// Mitsubishi GX Works2 project: Pneumalek2   PLC: Q03UDE

// global labels: Global1
VAR_GLOBAL
  Läge_0 AT M0 : BOOL;  (* Sensor *)
  Läge_1 AT M1 : BOOL;  (* Sensor *)
  Mag_sens AT M6 : BOOL;  (* Sensor *)
  Hämta_Mag : BOOL;
  Läge_2 AT M2 : BOOL;  (* Sensor *)
  Vrid_0 AT M3 : BOOL;  (* Sensor *)
  Vrid_1 AT M4 : BOOL;  (* Sensor *)
  Vrid_2 AT M5 : BOOL;  (* Sensor *)
  Kapacitiv AT M7 : BOOL;  (* Sensor *)
  Foto AT M8 : BOOL;  (* Sensor *)
  Induktiv AT M9 : BOOL;  (* Sensor *)
  Vakuum AT M10 : BOOL;  (* Sensor *)
  CylUppe AT M11 : BOOL;  (* Sensor *)
  CylNere AT M12 : BOOL;  (* Sensor *)
  Start AT M14 : BOOL;  (* Sensor *)
  Stopp AT M15 : BOOL;  (* Sensor *)
  PortalUt AT M17 : BOOL;  (* Actuator *)
  PortalIn AT M18 : BOOL;  (* Actuator *)
  VridHöger AT M19 : BOOL;  (* Actuator *)
  VridVänster AT M20 : BOOL;  (* Actuator *)
  CylNer AT M21 : BOOL;  (* Actuator *)
  CylUpp AT M22 : BOOL;  (* Actuator *)
  Sug : BOOL;
  Lämna_Sens : BOOL;
  Metall : BOOL;
  Vit : BOOL;
  Svart : BOOL;
  Sensor_Kopp : BOOL;
  Hämta_Sens : BOOL;
  LämnaMetall : BOOL;
  LämnaSvart : BOOL;
  LämnaVit : BOOL;
  Ejektor AT M23 : BOOL;  (* Actuator *)
  RESET : BOOL;
  ResetLägeP AT M16 : BOOL;  (* Sensor *)
  Portal : INT;
  Vrid : INT;
  PortalPos : INT;
  VridPos : INT;
  Hämta : BOOL;  (* Utan Last *)
  Lämna : BOOL;  (* Med Last *)
  Test_1 : BOOL;
  TestTimer1 : TON;
  TestTimer2 : TON;
  TestTimer3 : TON;
  TestTimer4 : TON;
  TestCount_1 : CTU;
  Testfunk1 : BOOL;
  TestTimer5 : TON;
  TestTimer6 : TON;
  TestTimer7 : TON;
  VridEQ : BOOL;
  PortalEQ : BOOL;
  Vänta_Sens : BOOL;
  TestM : BOOL;
  TestV : BOOL;
  TestS : BOOL;
  TestTimer8 : TON;
  TestTimer9 : TON;
  Timer7 : TON;
END_VAR

// task Task_01 (event TRUE, interval 0, priority 31): Sekvens, Applikation, testa

PROGRAM Sekvens
VAR
  Kör : BOOL;
END_VAR
(* structured ladder/FBD written out as ST: instructions are called as NAME(EN, inputs, outputs); _pN, _eN, _tN stand for wires *)
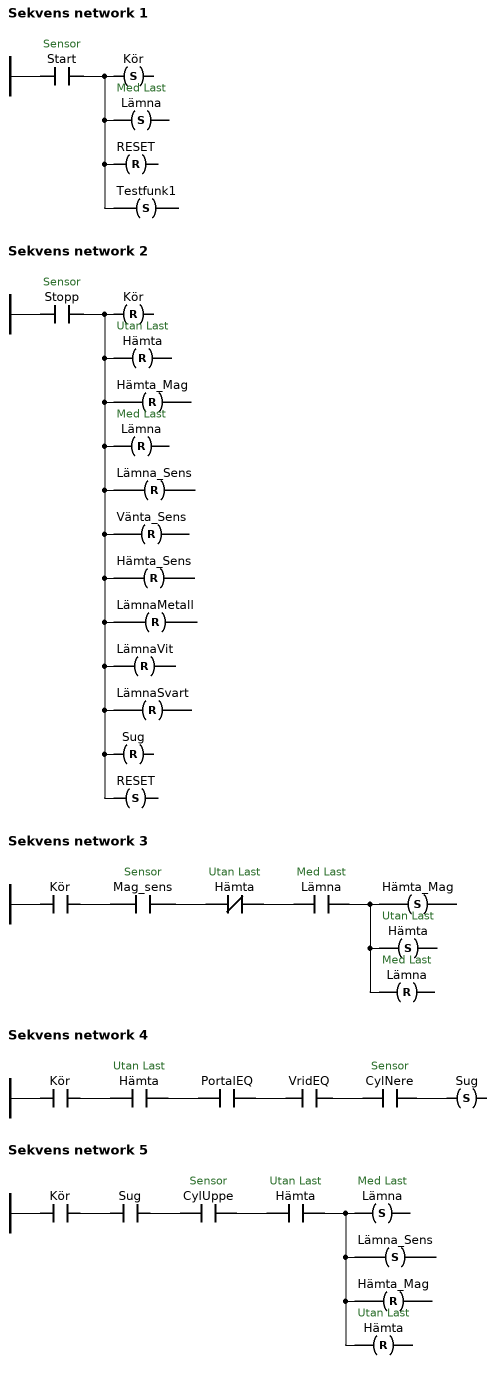
(* network 1 *)
SET(Start, Kör);
SET(Start, Lämna);
RST(Start, RESET);
SET(Start, Testfunk1);
(* network 2 *)
RST(Stopp, Kör);
RST(Stopp, Hämta);
RST(Stopp, Hämta_Mag);
RST(Stopp, Lämna);
RST(Stopp, Lämna_Sens);
RST(Stopp, Vänta_Sens);
RST(Stopp, Hämta_Sens);
RST(Stopp, LämnaMetall);
RST(Stopp, LämnaVit);
RST(Stopp, LämnaSvart);
RST(Stopp, Sug);
SET(Stopp, RESET);
(* network 3 *)
_p1 := Kör AND Mag_sens AND NOT Hämta AND Lämna;
SET(_p1, Hämta_Mag);
SET(_p1, Hämta);
RST(_p1, Lämna);
(* network 4 *)
SET(Kör AND Hämta AND PortalEQ AND VridEQ AND CylNere, Sug);
(* network 5 *)
_p1 := Kör AND Sug AND CylUppe AND Hämta;
SET(_p1, Lämna);
SET(_p1, Lämna_Sens);
RST(_p1, Hämta_Mag);
RST(_p1, Hämta);
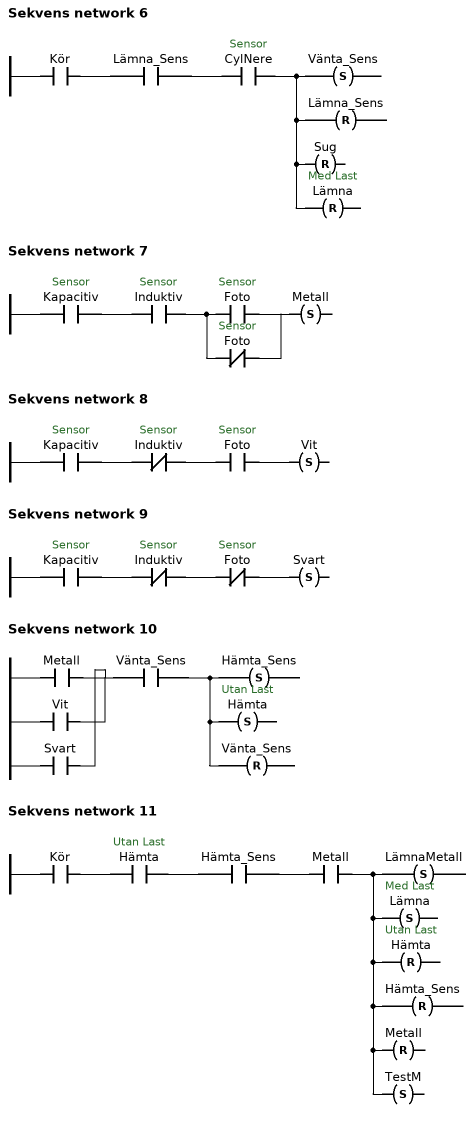
(* network 6 *)
_p1 := Kör AND Lämna_Sens AND CylNere;
SET(_p1, Vänta_Sens);
RST(_p1, Lämna_Sens);
RST(_p1, Sug);
RST(_p1, Lämna);
(* network 7 *)
_p1 := Kapacitiv AND Induktiv;
SET((_p1 AND Foto) OR (_p1 AND NOT Foto), Metall);
(* network 8 *)
SET(Kapacitiv AND NOT Induktiv AND Foto, Vit);
(* network 9 *)
SET(Kapacitiv AND NOT Induktiv AND NOT Foto, Svart);
(* network 10 *)
_p1 := (Metall OR Vit OR Svart) AND Vänta_Sens;
SET(_p1, Hämta_Sens);
SET(_p1, Hämta);
RST(_p1, Vänta_Sens);
(* network 11 *)
_p1 := Kör AND Hämta AND Hämta_Sens AND Metall;
SET(_p1, LämnaMetall);
SET(_p1, Lämna);
RST(_p1, Hämta);
RST(_p1, Hämta_Sens);
RST(_p1, Metall);
SET(_p1, TestM);
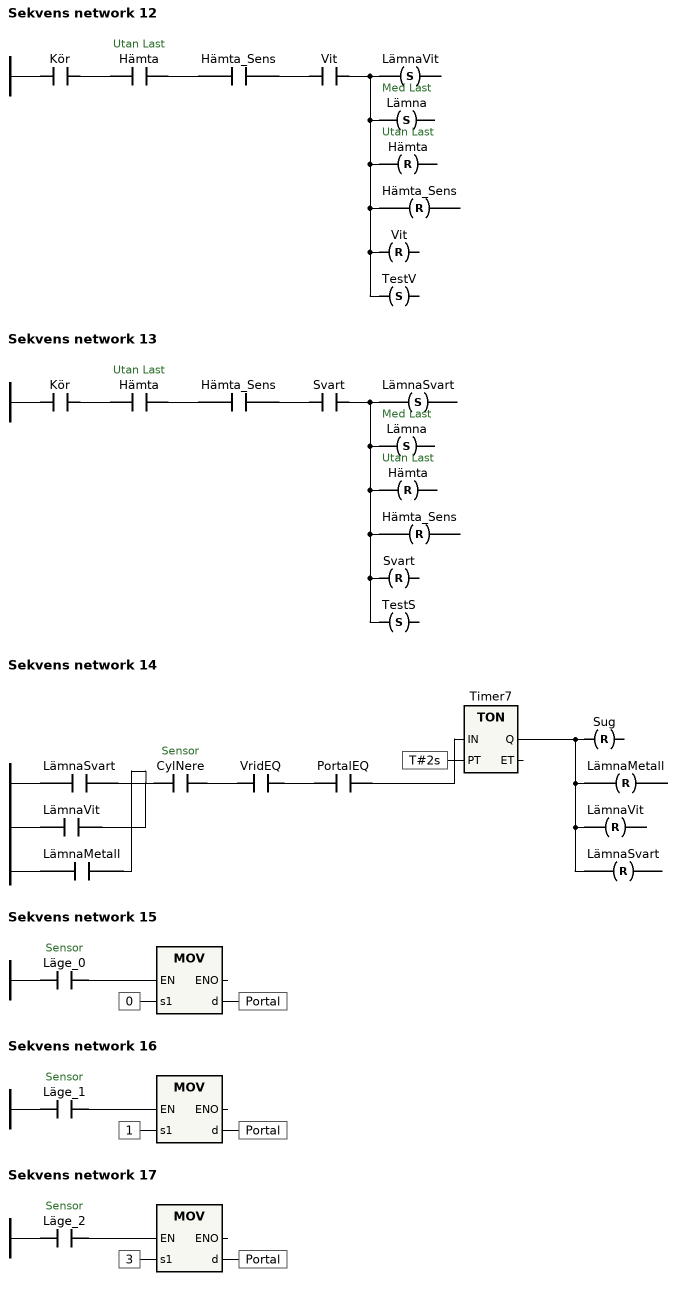
(* network 12 *)
_p1 := Kör AND Hämta AND Hämta_Sens AND Vit;
SET(_p1, LämnaVit);
SET(_p1, Lämna);
RST(_p1, Hämta);
RST(_p1, Hämta_Sens);
RST(_p1, Vit);
SET(_p1, TestV);
(* network 13 *)
_p1 := Kör AND Hämta AND Hämta_Sens AND Svart;
SET(_p1, LämnaSvart);
SET(_p1, Lämna);
RST(_p1, Hämta);
RST(_p1, Hämta_Sens);
RST(_p1, Svart);
SET(_p1, TestS);
(* network 14 *)
Timer7(IN := (((LämnaSvart OR LämnaVit OR LämnaMetall) AND CylNere) AND VridEQ) AND PortalEQ, PT := T#2s);
RST(Timer7.Q, Sug);
RST(Timer7.Q, LämnaMetall);
RST(Timer7.Q, LämnaVit);
RST(Timer7.Q, LämnaSvart);
(* network 15 *)
MOV(Läge_0, 0, Portal);
(* network 16 *)
MOV(Läge_1, 1, Portal);
(* network 17 *)
MOV(Läge_2, 3, Portal);
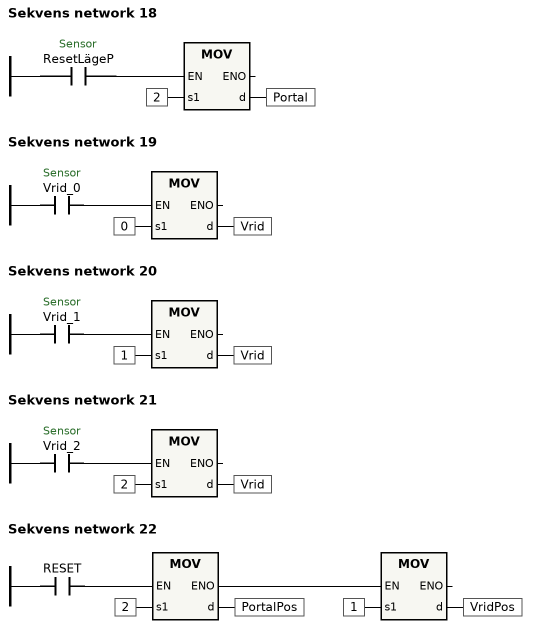
(* network 18 *)
MOV(ResetLägeP, 2, Portal);
(* network 19 *)
MOV(Vrid_0, 0, Vrid);
(* network 20 *)
MOV(Vrid_1, 1, Vrid);
(* network 21 *)
MOV(Vrid_2, 2, Vrid);
(* network 22 *)
_e1 := MOV(RESET, 2, PortalPos);
MOV(_e1, 1, VridPos);
END_PROGRAM

PROGRAM Applikation
VAR
  RESET1 : BOOL;
  RESET2 : BOOL;
  RESET3 : BOOL;
  RESET4 : BOOL;
  Timer1 : TON;
  Timer2 : TON;
  Timer3 : TON;
END_VAR
(* structured ladder/FBD written out as ST: instructions are called as NAME(EN, inputs, outputs); _pN, _eN, _tN stand for wires *)
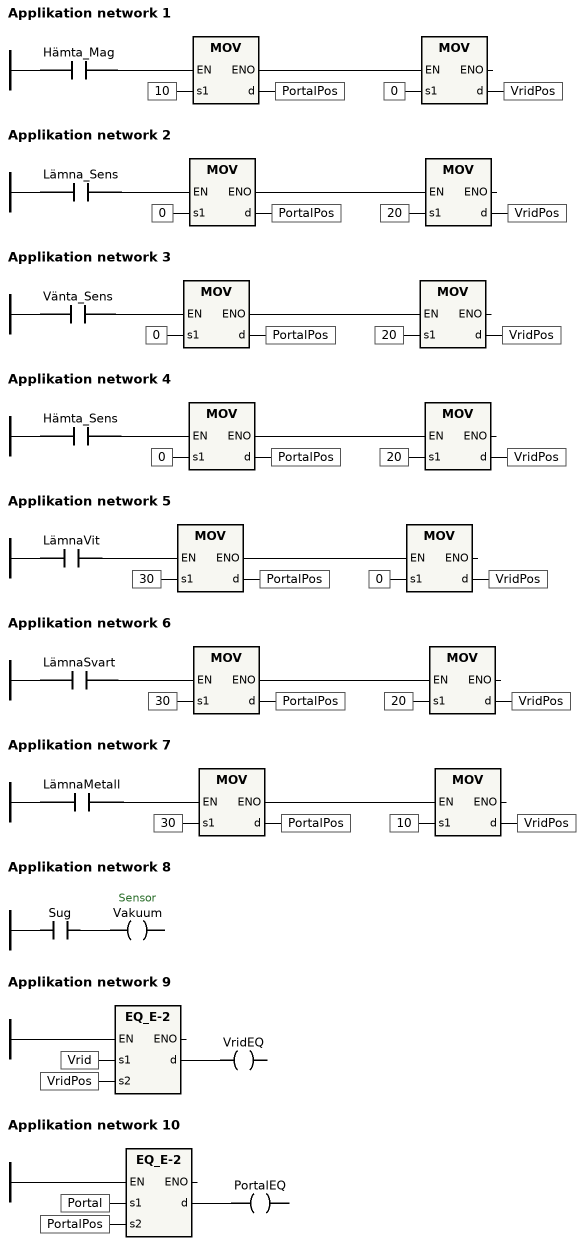
(* network 1 *)
_e1 := MOV(Hämta_Mag, 10, PortalPos);
MOV(_e1, 0, VridPos);
(* network 2 *)
_e1 := MOV(Lämna_Sens, 0, PortalPos);
MOV(_e1, 20, VridPos);
(* network 3 *)
_e1 := MOV(Vänta_Sens, 0, PortalPos);
MOV(_e1, 20, VridPos);
(* network 4 *)
_e1 := MOV(Hämta_Sens, 0, PortalPos);
MOV(_e1, 20, VridPos);
(* network 5 *)
_e1 := MOV(LämnaVit, 30, PortalPos);
MOV(_e1, 0, VridPos);
(* network 6 *)
_e1 := MOV(LämnaSvart, 30, PortalPos);
MOV(_e1, 20, VridPos);
(* network 7 *)
_e1 := MOV(LämnaMetall, 30, PortalPos);
MOV(_e1, 10, VridPos);
(* network 8 *)
Vakuum := Sug;
(* network 9 *)
EQ_E(TRUE, Vrid, VridPos, _t1);
VridEQ := _t1;
(* network 10 *)
EQ_E(TRUE, Portal, PortalPos, _t1);
PortalEQ := _t1;
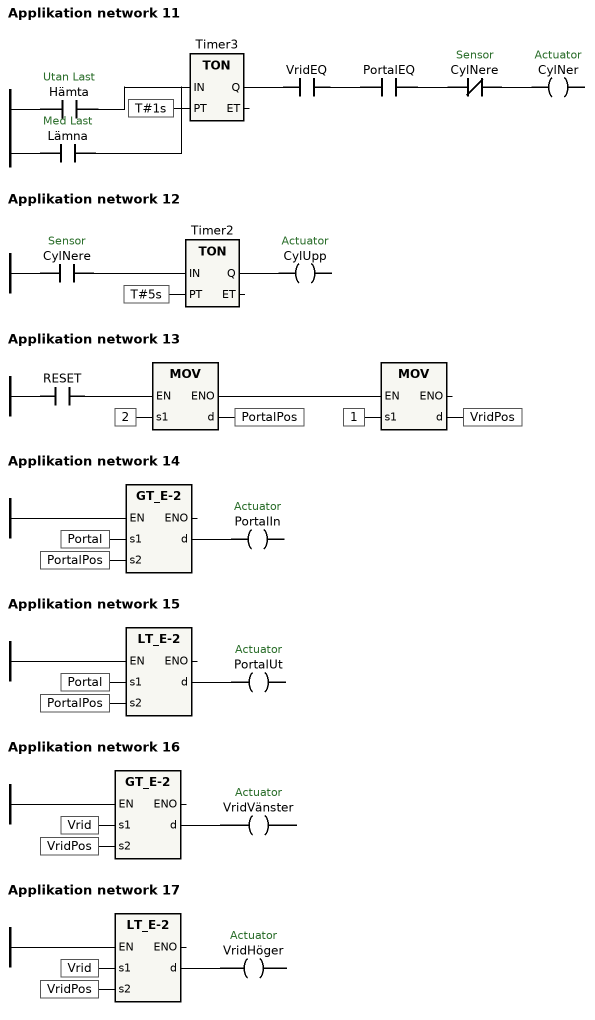
(* network 11 *)
Timer3(IN := Hämta OR Lämna, PT := T#1s);
CylNer := Timer3.Q AND VridEQ AND PortalEQ AND NOT CylNere;
(* network 12 *)
Timer2(IN := CylNere, PT := T#5s);
CylUpp := Timer2.Q;
(* network 13 *)
_e1 := MOV(RESET, 2, PortalPos);
MOV(_e1, 1, VridPos);
(* network 14 *)
GT_E(TRUE, Portal, PortalPos, _t1);
PortalIn := _t1;
(* network 15 *)
LT_E(TRUE, Portal, PortalPos, _t1);
PortalUt := _t1;
(* network 16 *)
GT_E(TRUE, Vrid, VridPos, _t1);
VridVänster := _t1;
(* network 17 *)
LT_E(TRUE, Vrid, VridPos, _t1);
VridHöger := _t1;
END_PROGRAM

PROGRAM testa
VAR
  TestCounter1 : CTU;
  TestCounter2 : CTU;
  TestCounter3 : CTU;
END_VAR
(* structured ladder/FBD written out as ST: instructions are called as NAME(EN, inputs, outputs); _pN, _eN, _tN stand for wires *)
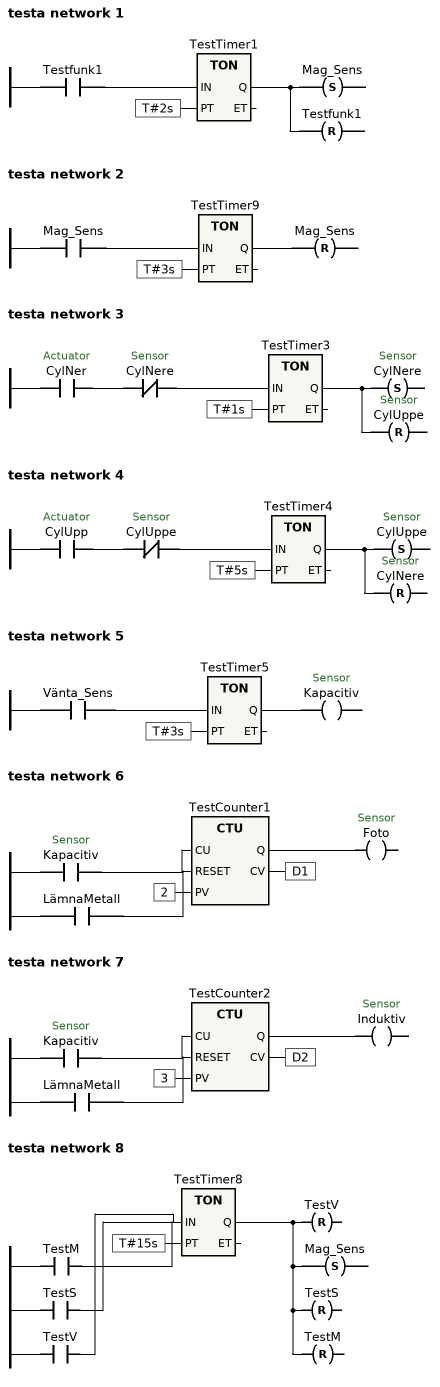
(* network 1 Test1: *)
TestTimer1(IN := Testfunk1, PT := T#2s);
SET(TestTimer1.Q, Mag_Sens);
RST(TestTimer1.Q, Testfunk1);
(* network 2 Test2: *)
TestTimer9(IN := Mag_Sens, PT := T#3s);
RST(TestTimer9.Q, Mag_Sens);
(* network 3 Test3: *)
TestTimer3(IN := CylNer AND NOT CylNere, PT := T#1s);
SET(TestTimer3.Q, CylNere);
RST(TestTimer3.Q, CylUppe);
(* network 4 Test3_2: *)
TestTimer4(IN := CylUpp AND NOT CylUppe, PT := T#5s);
SET(TestTimer4.Q, CylUppe);
RST(TestTimer4.Q, CylNere);
(* network 5 Test4: *)
TestTimer5(IN := Vänta_Sens, PT := T#3s);
Kapacitiv := TestTimer5.Q;
(* network 6 Test4_2: *)
TestCounter1(CU := Kapacitiv, RESET := LämnaMetall, PV := 2, CV => D1);
Foto := TestCounter1.Q;
(* network 7 Test4_3: *)
TestCounter2(CU := Kapacitiv, RESET := LämnaMetall, PV := 3, CV => D2);
Induktiv := TestCounter2.Q;
(* network 8 Test5: *)
TestTimer8(IN := TestM OR TestS OR TestV, PT := T#15s);
RST(TestTimer8.Q, TestV);
SET(TestTimer8.Q, Mag_Sens);
RST(TestTimer8.Q, TestS);
RST(TestTimer8.Q, TestM);
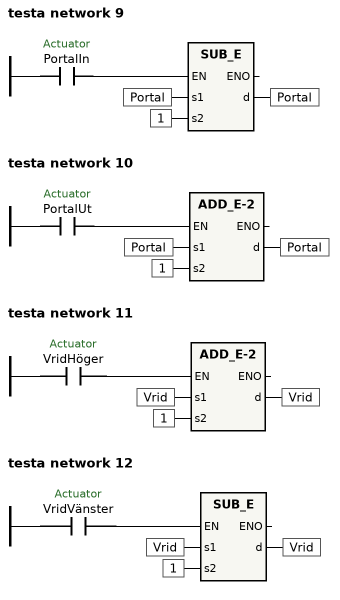
(* network 9 Test9_1: *)
SUB_E(PortalIn, Portal, 1, Portal);
(* network 10 Test9_2: *)
ADD_E(PortalUt, Portal, 1, Portal);
(* network 11 Test9_3: *)
ADD_E(VridHöger, Vrid, 1, Vrid);
(* network 12 Test9_4: *)
SUB_E(VridVänster, Vrid, 1, Vrid);
END_PROGRAM
